{attribute addProperty BoxType "EP7402-0057-0017"}
{attribute addProperty Id "ControlAT %Q*Control_01CFC91D162"}
{attribute addProperty CRC "3571864908"}
{attribute addProperty SizeInBites "16"}
{attribute addProperty SizeInBytes "2"}
TYPE STM_Control_Channel_D4E6554C :
STRUCT
	{attribute addProperty Name "Control"}
	Control AT %Q* : Control_01CFC91D;
END_STRUCT
END_TYPE

(* stored: Version 1.2.0.0, ProductVersion 3.1.4024.9
   DUT STM_Control_Channel_D4E6554C: Id {f11eae16-d994-4667-8a9c-be162f366686} *)
